FUNCTION_BLOCK WrappableList
VAR_INPUT
END_VAR
VAR_OUTPUT
	count : UINT;
	_typeClass : __SYSTEM.TYPE_CLASS; // Type of data object - primitives or Userdef
	_classSize : DINT; // Size of data object - useful to check type of Userdef typeclass
END_VAR
VAR
	head : POINTER TO Node := NULL;
	tail : POINTER TO Node := NULL;
END_VAR

METHOD PROTECTED _Append : REFERENCE TO WrappableList
VAR_INPUT
	data : ANY;
END_VAR
VAR
	new : POINTER TO Node;
END_VAR
_Append REF= THIS^;

IF NOT IsTypeClassCorrect(data) THEN
	RETURN;
END_IF
SetTypeClass(data);

new := __NEW(Node);
new^.data := __NEW(BYTE, classSize);
MEMCPY(new^.data, data.pValue, classSize);
new^.next := NULL;

IF head = NULL THEN
	head := new;
	tail := new;
ELSE
	tail^.next := new;
	tail := tail^.next;
END_IF
count := count + 1;
END_METHOD


METHOD PROTECTED _Get : REFERENCE TO WrappableList
VAR_INPUT
	// indexing from end allowed
	// index = 0 returns first element
	// index = 1 returns seconds element
	// index = -1 returns last element
	// index = -2 return before-last element
	index : INT;
	destinationVariable : ANY;
END_VAR
VAR
	current : POINTER TO Node := NULL;
	getIndex : INT;
	i : INT;
END_VAR

IF NOT IsTypeClassCorrect(destinationVariable) THEN
	RETURN;
END_IF;

IF head = NULL THEN
	RETURN;
END_IF;

// Calculate actual index in List
getIndex := (count * BOOL_TO_INT(index < 0)) + index;

// Return 0 for invalid indexes
IF 	(getIndex >= count) OR	// Indexing from begin begins with 0
	(getIndex < 0) // Indexing from end begins with -1
THEN
	RETURN;
END_IF


current := head;
FOR i := 1 TO getIndex DO // we already got head in previous line, that's why it's from 1
	IF current^.next = NULL THEN
		RETURN;
	END_IF
	current := current^.next;
END_FOR
MEMMOVE(destinationVariable.pValue, current^.data, classSize);
END_METHOD


//{attribute 'monitoring' := 'call'}
// Size of data object - useful to check type of Userdef typeclass
PROPERTY classSize : DINT
GET

classSize := _classSize;
END_GET
SET // PRIVATE

_classSize := classSize;
END_SET
END_PROPERTY

// Inserts new element into given index. Negative indexing is supported
METHOD Insert : REFERENCE TO WrappableList
VAR_INPUT
	(*
		0 = Prepend;
		1 = Insert into second position;
		-2 = Insert into second position from end;
		-1 = Append;
	*)
	index : INT;
	data : ANY;
END_VAR
VAR
	new : POINTER TO Node;
	current : POINTER TO Node;
	insertIndex : INT;
	i : INT;
END_VAR

Insert REF= THIS^;

IF NOT IsTypeClassCorrect(data) THEN
	RETURN;
END_IF
SetTypeClass(data);

new := __NEW(Node);
new^.data := __NEW(BYTE, classSize);
MEMCPY(new^.data, data.pValue, classSize);

// Calculate actual index in List
insertIndex := ((count + 1) * BOOL_TO_INT(index < 0)) + index;

IF insertIndex >= count // Index too high -> append to end
THEN
	_Append(data);
	RETURN;
ELSIF insertIndex <= 0 // Index too high from the end -> prepend to beginning
THEN
	Prepend(data);
	RETURN;
END_IF

current := head;
FOR i := 1 TO insertIndex - 1 DO
	current := current^.next;
END_FOR
new^.next := current^.next;
current^.next := new;
count := count + 1;
END_METHOD


METHOD IsEmpty : BOOL
VAR_INPUT
END_VAR

IsEmpty := head = NULL;
END_METHOD


METHOD IsTypeClassCorrect : BOOL
VAR_INPUT
	CheckedVariable : ANY;
END_VAR

IF classSize = 0 THEN
	IsTypeClassCorrect := TRUE;
	RETURN;
END_IF
IsTypeClassCorrect := typeClass = CheckedVariable.TypeClass AND classSize = CheckedVariable.diSize;
END_METHOD


// Pushes data to the beginning of the list
METHOD Prepend : REFERENCE TO WrappableList
VAR_INPUT
	data : ANY;
END_VAR
VAR
	new : POINTER TO Node;
END_VAR

Prepend REF= THIS^;

IF NOT IsTypeClassCorrect(data) THEN
	RETURN;
END_IF
SetTypeClass(data);

new := __NEW(Node);
new^.data := __NEW(BYTE, classSize);
MEMCPY(new^.data, data.pValue, classSize);
new^.next := head;

IF head = NULL THEN
	head := new;
	tail := new;
ELSE
	head := new;
END_IF
count := count + 1;
END_METHOD


METHOD Remove : REFERENCE TO WrappableList;
VAR_INPUT
	index : INT;
END_VAR
VAR
	current : POINTER TO Node := NULL;
	removeIndex : INT;	
	nodeToRemove : POINTER TO Node;
	i : INT;
END_VAR

Remove REF= THIS^;

IF head = NULL THEN
	RETURN;
END_IF;

// Calculate actual index in List
removeIndex := (count * BOOL_TO_INT(index < 0)) + index; 

// Cancel removal for invalid indexes
IF 	(removeIndex >= count) OR // Indexing from begin begins with 0
	(removeIndex < 0) // Indexing from end begins with -1
THEN
	RETURN;
END_IF

IF removeIndex = 0 THEN
	nodeToRemove := head;
	head := head^.next;
ELSE
	current := head;
	FOR i := 1 TO removeIndex - 1 DO
		current := current^.next;
	END_FOR
	nodeToRemove := current^.next;
	current^.next := current^.next^.next;
END_IF
IF nodeToRemove = tail THEN
	tail := current;
END_IF
__DELETE(nodeToRemove^.data);
__DELETE(nodeToRemove);
count := count - 1;
END_METHOD


METHOD RemoveAll : REFERENCE TO WrappableList
VAR_INPUT
END_VAR

WHILE head <> NULL DO
	Remove(0);
END_WHILE
END_METHOD


METHOD SetTypeClass : BOOL
VAR_INPUT
	ReferenceVariable : ANY; // Pass any variable of your chosen type. It will only be used to obtain data type
END_VAR

IF classSize = 0 THEN
	typeClass := ReferenceVariable.TypeClass;
	classSize := ReferenceVariable.diSize;
	SetTypeClass := TRUE;
END_IF
END_METHOD


//{attribute 'monitoring' := 'call'}
// Type of data object - primitives or Userdef
PROPERTY typeClass : __SYSTEM.TYPE_CLASS
GET

typeClass := _typeClass;
END_GET
SET // PRIVATE

_typeClass := typeClass;
END_SET
END_PROPERTY

END_FUNCTION_BLOCK

(* stored: Version 1.1.0.1, ProductVersion 3.1.4024.11
   POU WrappableList: Id {ca08b2fb-2d23-4b3e-81bb-a2facb2a8425}, SpecialFunc None
   Method _Append: Id {40e96914-b8be-4eb1-83bd-e01089932ae8}
   Method _Get: Id {c2722b16-7c99-41ac-a740-753b89560dea}
   Property classSize: Id {472807a7-4887-42a4-9772-3a0fa6f7a368}
   Get Get: Id {11a13790-f3d1-42c8-bed6-f7e32953bc59}
   Set Set: Id {607e393b-3979-4efc-8fe4-6059ba11c1c7}
   Method Insert: Id {dc1fed3d-f702-4622-bcf1-8e347a9d306e}
   Method IsEmpty: Id {effa7d14-2ac9-4336-9502-f0e2f8f66119}
   Method IsTypeClassCorrect: Id {57ad85de-1bf2-4568-88e8-b597de22c725}
   Method Prepend: Id {a005bd10-c0a4-428e-b47d-b3a0bae09a55}
   Method Remove: Id {86e69ae2-79e1-49a0-be8b-fbc89ffa93eb}
   Method RemoveAll: Id {7b77c637-bdf7-4ab8-b391-bbc2186a0a44}
   Method SetTypeClass: Id {1bd4d152-eddc-424a-a539-895a22ed9f1e}
   Property typeClass: Id {47310767-7ddb-473e-ae58-91644eca8bba}
   Get Get: Id {6e72db4f-0187-4d25-9772-2f57b7c9c04e}
   Set Set: Id {276b8d61-c05d-441f-baa7-50c671d7c0fa} *)
